# EPICS substitutions: myexampleApp/Db/user.substitutions
# Example substitutions file

file "dbExample1.db" {
    { user = "jhlee" }
}

file dbExample2.db {
    pattern { user, no, scan }
        { "jhlee", 1, "1 second" }
        { "jhlee", 2, "2 second" }
        { "jhlee", 3, "5 second" }
}
